PROGRAM MAIN
VAR
	bInit: BOOL := TRUE;
	fbSocketCloseAll: FB_SocketCloseAll; 
	bSocketCloseError: BOOL;
	nSocketCloseError: UDINT;
	
	fbTcpClient1					: FB_TCPClient;
		sClient1SendData			: STRING(255);
		nServer1Port				: UDINT 				:= 2010;
		sServer1Host				: T_IPv4Addr 			:= '';
		bStartClient1Communication	: BOOL 					:= FALSE;
		tClient1CycleTime			: TIME 					:= T#0.5S;
		bClient1SendTrigger			: BOOL;
		bClient1Connected			: BOOL;
		sClient1ReceivedData		: STRING(255);
		bClient1Busy				: BOOL;
		bClientError1				: BOOL;
		nClient1ErrorID1			: UDINT;		
		
	fbTcpEchoServer1				: FB_TCPServer;
		sServerReceivedData			: STRING(255);
		bStartServer1Communication	: BOOL 					:= TRUE;
		bServer1Connected			: BOOL;
		sServerData					: STRING(255);
		bServer1Busy				: BOOL;
		bServer1Error				: BOOL;
		nServer1ErrorID				: UDINT;
	
	bAutogenerateData				: BOOL 					:= TRUE;
	fbTimer1						: TON;
	nCnt							: UDINT;
	
// Optional second Client and Server
(*	fbTcpClient2					: FB_TCPClient;
		sClient2SendData			: STRING(255)			:= 'TestString123';
		sClient2ReceivedData		: STRING(255);			
	fbTcpServer2					: FB_TCPServer;
		sServer2Data				: STRING(255); *)
END_VAR

IF bInit THEN 				// Init Step to close all sockets after login PLC with  downlaod
	fbSocketCloseAll(
		sSrvNetId:= '', 
		bExecute:= TRUE, 
		tTimeout:= T#3S, 
		bBusy=> , 
		bError=> bSocketCloseError, 
		nErrId=> nSocketCloseError);
	IF NOT (fbSocketCloseAll.bBusy OR fbSocketCloseAll.bError) THEN
		bInit := FALSE;
		fbSocketCloseAll(bExecute:= FALSE);
	END_IF
ELSE
	
	fbTcpClient1(
		nRemotePort:= nServer1Port, 								// Server port
		sRemoteHost:= sServer1Host, 								// Server IP (empty for local communication)
		bStartCommunication:= bStartClient1Communication, 			// Start communication, when FALSE, connection is closed
		sSendData:= sClient1SendData, 								// Data that are sent to the server
		tCycleTimeSend:= (*tClient1CycleTime*), 					// TimeInterval for cyclic sending
		bSendTrigger:= ,											// Trigger to send one telegramm manually 
		bConnected => bClient1Connected,							// Switches to TRUE when Client is connected to a server
		sReceivedData=> sClient1ReceivedData,						// Data that are received
		bBusy=> bClient1Busy, 
		bError=> bClientError1, 
		nErrorID=> nClient1ErrorID1, ); 
	
	IF bAutogenerateData AND bClient1Connected THEN
		fbTimer1(IN:= NOT fbTimer1.Q, PT:= tClient1CycleTime, Q=> , ET=> );
		IF fbTimer1.Q  THEN
			sClient1SendData := Concat('TestString No.', UDINT_TO_STRING(nCnt));
			fbTcpClient1.bSendTrigger := TRUE;
			nCnt := nCnt + 1;
		ELSE
			fbTcpClient1.bSendTrigger := FALSE;
		END_IF
	END_IF 
		
	fbTcpEchoServer1(
		sLocalHost:= '192.168.1.4', 											// Server IP Adress
		nLocalPort:= nServer1Port, 									// Server port
		bStartCommunication:= bStartServer1Communication, 			// Allow Client-connection or close connection
		bConnected => bServer1Connected,							// Client connection is valid
		sSendData => sServerData,
		bBusy=> bServer1Busy, 
		bError=> bServer1Error, 
		nErrorID=> nServer1ErrorID);
	
	// Optional second Client and Server
	
(*	fbTcpClient2(
		sRemoteHost:= '', 
		nRemotePort:= 12001, 
		sSendData:= sClient2SendData, 
		bStartCommunication:= TRUE, 
		tCycleTimeSend:= T#2S, 
		bSendTrigger:= ,
		bConnected => , 
		sReceivedData=> sClient2ReceivedData, 
		nErrorID=> , 
		bError=> , 
		bBusy=> );
		
	fbTcpServer2(
		sLocalHost:= '', 
		nLocalPort:= 12001, 
		bStartCommunication:= TRUE, 
		sSendData => sServer2Data, 
		bBusy=> , 
		bError=> , 
		nErrorID=> ); *)
END_IF

END_PROGRAM

(* stored: Version 1.1.0.1, ProductVersion 3.1.4024.12
   POU MAIN: Id {572507de-a44a-4a7e-b7eb-52f2373576ea}, SpecialFunc None *)
